(****************************************************************
NAME:			FB_LedShow
DATA:			2017.2.16
VERSION:		1.0.0
DESCRIPTION:	FB_LedShow
HISTORY:
				2017.2.16 	NEW

***************************************************************)
FUNCTION_BLOCK FB_LedShow
VAR_INPUT
	Error:BOOL;
	Run:BOOL;
END_VAR
VAR_OUTPUT
	LedStatus:DINT;
END_VAR
VAR
END_VAR

IF Run THEN
	Led_Run:=TRUE;
	Led_Error:=FALSE;
	LedStatus:=1;
END_IF

IF Error THEN
	Led_Run:=FALSE;
	Led_Error:=TRUE;
	LedStatus:=0;
END_IF

END_FUNCTION_BLOCK

(* stored: Version 1.1.0.1, ProductVersion 3.1.4024.6
   POU FB_LedShow: Id {18e4c288-3d16-46ba-b7ee-e99ba52b271b}, SpecialFunc None *)
